// TwinCAT 3 PLC project mobject_enumerable
// Title: mobject-enumerable
// Company: mobject
// Author: mobject dev team
// ProjectVersion: 1.2.0
// ProgramVersion: 3.1.4024.0
// libraries:
//   Tc2_System, * (Beckhoff Automation GmbH)
//   mobject-disposable,1.1.1,mobject
// project tree:
//   Interfaces/Enumerators/ I_ForwardEnumerator.TcIO, I_KeyValueForwardEnumerator.TcIO
//   Interfaces/ I_Enumerable.TcIO, I_KeyValueEnumerable.TcIO

// ---- Interfaces/Enumerators/I_ForwardEnumerator.TcIO
INTERFACE I_ForwardEnumerator EXTENDS I_Disposable

PROPERTY PUBLIC IsValid : BOOL
GET
END_GET
END_PROPERTY

METHOD PUBLIC MoveNext : BOOL
END_METHOD

METHOD PUBLIC Reset
END_METHOD

METHOD PUBLIC TryGet : BOOL;
VAR_INPUT
    Destination : ANY;
END_VAR
END_METHOD

METHOD PUBLIC TryGetTo : BOOL;
VAR_INPUT
    DestinationAddress : PVOID;
    DestinationSize : UDINT;
END_VAR
END_METHOD

END_INTERFACE

// ---- Interfaces/Enumerators/I_KeyValueForwardEnumerator.TcIO
INTERFACE I_KeyValueForwardEnumerator EXTENDS I_ForwardEnumerator

PROPERTY Key : T_MAXSTRING
GET
END_GET
END_PROPERTY

END_INTERFACE

// ---- Interfaces/I_Enumerable.TcIO
INTERFACE I_Enumerable EXTENDS __SYSTEM.IQueryInterface

METHOD PUBLIC GetEnumerator : I_ForwardEnumerator
END_METHOD

END_INTERFACE

// ---- Interfaces/I_KeyValueEnumerable.TcIO
INTERFACE I_KeyValueEnumerable EXTENDS __SYSTEM.IQueryInterface

METHOD PUBLIC GetKeyValueEnumerator : I_KeyValueForwardEnumerator
END_METHOD

END_INTERFACE
